(*
	Simple solutions for the exercices of the book 
	Collection of Exercises for PLC Programming
	by Tom Mejer Antonson
	ISBN: 978-87-4305-780-2
*)
PROGRAM MAIN
VAR
END_VAR

//LogicalCircuits();
//Safety();
//LogicAndCounters();
//Timers();
AnalogSignals();
//AppliedMathematics();
//Arrays();
//FunctionsAndFunctionBlocks();
//StringsAndStructs();
//ComplexExercises();

END_PROGRAM

(* stored: Version 1.1.0.1
   POU MAIN: Id {2fad4f42-d39c-4c01-a8b8-3ea2910d0ceb}, SpecialFunc None *)
